// TIA Portal project "Machines ON OFF with Pushbutton Switch" (V17)
// Machines ON OFF with Pushbutton Switch
// When Switch (pushbutton) is turned ON (pressed) and then turned OFF (released), then Machine 1 will be ON.
// And then, when Switch (pushbutton) is turned ON (pressed) and then turned OFF (released), then Machine 1 will be OFF and Machine 2 will be ON.
// And then, when Switch (pushbutton) is turned ON (pressed) and then turned OFF (released), then Machine 2 will be OFF and Machine 3 will be ON.

(* hardware
DEVICE "S7-1200 station_1"  S7-1200 Station
   slot 0: "Rack_0"  S7-1200 Rack  Rack  V1.0
   slot 1: "PLC_1"  CPU 1212C AC/DC/Rly  6ES7 212-1BE40-0XB0  V4.5
*)

// ===== PLC "PLC_1"  CPU 1212C AC/DC/Rly =====

VAR_GLOBAL   // PLC tag table "Default tag table"
   "Pushbutton" AT %I0.0 : Bool;
   "Machine 1" AT %Q0.0 : Bool;
   "Machine 2" AT %Q0.1 : Bool;
   "Machine 3" AT %Q0.2 : Bool;
   "Tag_1" AT %M0.0 : Bool;
   "Tag_2" AT %M0.1 : Bool;
   "Tag_3" AT %M0.2 : Bool;
   "Tag_4" AT %M0.3 : Bool;
END_VAR

ORGANIZATION_BLOCK "Main"   // OB1, LAD, ProgramCycle
TITLE = "Main Program Sweep (Cycle)"
{ S7_Optimized_Access := 'TRUE' }
VERSION : 0.1
   VAR_INPUT
      Initial_Call : Bool;   // Initial call of this OB
      Remanence : Bool;   // =True, if remanent data are available
   END_VAR
BEGIN

REGION Network 1
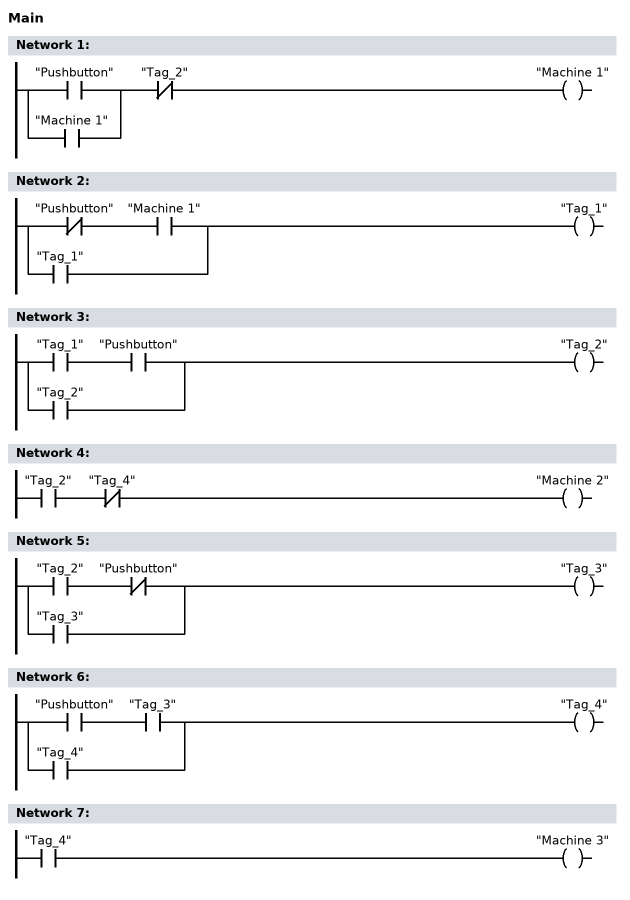
   RUNG wire#powerrail
      Contact( "Pushbutton" )
      wire#w1
      I_Contact( "Tag_2" )
      Coil( "Machine 1" )
   END_RUNG
   RUNG wire#powerrail
      Contact( "Machine 1" )
   END_RUNG wire#w1
   // the same network as SCL:
   "Machine 1" := ("Pushbutton" OR "Machine 1") AND NOT "Tag_2";
END_REGION

REGION Network 2
   RUNG wire#powerrail
      I_Contact( "Pushbutton" )
      Contact( "Machine 1" )
      wire#w1
      Coil( "Tag_1" )
   END_RUNG
   RUNG wire#powerrail
      Contact( "Tag_1" )
   END_RUNG wire#w1
   // the same network as SCL:
   "Tag_1" := (NOT "Pushbutton" AND "Machine 1") OR "Tag_1";
END_REGION

REGION Network 3
   RUNG wire#powerrail
      Contact( "Tag_1" )
      Contact( "Pushbutton" )
      wire#w1
      Coil( "Tag_2" )
   END_RUNG
   RUNG wire#powerrail
      Contact( "Tag_2" )
   END_RUNG wire#w1
   // the same network as SCL:
   "Tag_2" := ("Tag_1" AND "Pushbutton") OR "Tag_2";
END_REGION

REGION Network 4
   RUNG wire#powerrail
      Contact( "Tag_2" )
      I_Contact( "Tag_4" )
      Coil( "Machine 2" )
   END_RUNG
   // the same network as SCL:
   "Machine 2" := "Tag_2" AND NOT "Tag_4";
END_REGION

REGION Network 5
   RUNG wire#powerrail
      Contact( "Tag_2" )
      I_Contact( "Pushbutton" )
      wire#w1
      Coil( "Tag_3" )
   END_RUNG
   RUNG wire#powerrail
      Contact( "Tag_3" )
   END_RUNG wire#w1
   // the same network as SCL:
   "Tag_3" := ("Tag_2" AND NOT "Pushbutton") OR "Tag_3";
END_REGION

REGION Network 6
   RUNG wire#powerrail
      Contact( "Pushbutton" )
      Contact( "Tag_3" )
      wire#w1
      Coil( "Tag_4" )
   END_RUNG
   RUNG wire#powerrail
      Contact( "Tag_4" )
   END_RUNG wire#w1
   // the same network as SCL:
   "Tag_4" := ("Pushbutton" AND "Tag_3") OR "Tag_4";
END_REGION

REGION Network 7
   RUNG wire#powerrail
      Contact( "Tag_4" )
      Coil( "Machine 3" )
   END_RUNG
   // the same network as SCL:
   "Machine 3" := "Tag_4";
END_REGION
END_ORGANIZATION_BLOCK